FUNCTION_BLOCK FB_VALVE_RELAY

VAR
// EL2624 Relayu Logic Here
	{attribute 'pytmc' := 'pv: XBD:N2:VRC:01'}
	{attribute 'TcLinkTo' := 'TIID^Device 1 (EtherCAT)^Term 1 (EK1200)^Term 5 (EL2624)^Channel 1^Output'}
	rawOutputRelayChan1 AT %Q*: BOOL;

	{attribute 'pytmc' := 'pv: XBD:N2:VRC:02'}
	{attribute 'TcLinkTo' := 'TIID^Device 1 (EtherCAT)^Term 1 (EK1200)^Term 5 (EL2624)^Channel 2^Output'}
	rawOutputRelayChan3 AT %Q*: BOOL;
	
	{attribute 'TcLinkTo' := 'TIID^Device 1 (EtherCAT)^Term 1 (EK1200)^Term 6 (EL1004)^Channel 1^Input'}
	bCloseRBV AT %I* : BOOL;
	{attribute 'TcLinkTo' := 'TIID^Device 1 (EtherCAT)^Term 1 (EK1200)^Term 6 (EL1004)^Channel 2^Input'}
	bOpenRBV AT %I* : BOOL;
	{attribute 'TcLinkTo' := 'TIID^Device 1 (EtherCAT)^Term 1 (EK1200)^Term 6 (EL1004)^Channel 3^Input'}
	bMovingRBV AT %I* : BOOL;
	
	b_open : BOOL;
	b_complete: BOOL;
	iState: INT; // init = 0, nominsl = 1, timer = 2
	iPosState: INT; // 0 = Moving, 1 = CLOSED; 2 = OPEN
	bPrevPos : BOOL;
	bMaintenanceMode: BOOL;


END_VAR

VAR_INPUT
END_VAR
VAR_OUTPUT
END_VAR
VAR
	fbValveTimer : TON;
    fbCloseValveTimer : TOF;
END_VAR


fbValveTimer(IN:=TRUE); //RESTART TIMER

CASE iState OF
    0: // INIT
    fbValveTimer(IN:=FALSE); //RESTART TIMER
    iState := 1;

    1: // NOMINAL
	IF b_open THEN
    	rawOutputRelayChan1 := FALSE;
    	rawOutputRelayChan3 := TRUE;
	ELSE
    	rawOutputRelayChan1 := TRUE;
    	rawOutputRelayChan3 := FALSE;
	END_IF
	
	
	IF bMovingRBV THEN
		b_complete := FALSE;
	ELSE
		b_complete := TRUE;
		IF bCloseRBV THEN
			iPosState := 1;
		ELSIF bOpenRBV THEN
			iPosState := 2;
		END_IF
	END_IF
	// tick timer check if elapsed
 
	IF fbValveTimer.Q THEN
		iState := 2;
	END_IF
	
	2: // TIMER
	IF iPosState = 2 THEN // if closed
    	rawOutputRelayChan1 := TRUE;
    	rawOutputRelayChan3 := FALSE;
	ELSIF iPosState = 1 THEN // if open close
    	rawOutputRelayChan1 := FALSE;
    	rawOutputRelayChan3 := TRUE;
	END_IF	
	IF bMovingRBV THEN
		b_complete := FALSE;
	ELSE
		b_complete := TRUE;
		iState := 0; // go to 0 to restart the timer
	END_IF
END_CASE

END_FUNCTION_BLOCK

(* stored: Version 1.1.0.1, ProductVersion 3.1.4024.11
   POU FB_VALVE_RELAY: Id {e2531ff2-ea72-4542-bd8f-7299f2dc48b9}, SpecialFunc None *)
